{attribute 'GeneratedUsingTerminal: EK1100-0000-0018'}
{attribute addProperty BoxType "EK1100-0000-0018"}
{attribute addProperty Id "Beckhoff_EPP7xxxEK1122Beckhoff_EPP7xxxEK1122_6A0F0FE8478"}
{attribute addProperty CRC "1759912252"}
{attribute addProperty Size "478"}
TYPE Beckhoff_EPP7xxx_68E6213C EXTENDS EK1100_1FC0878B :
STRUCT
	{attribute addProperty Name "Beckhoff_EPP7xxxEK1122"}
	{attribute addProperty PreviousPort "Beckhoff EPP7xxx : B"}
	Beckhoff_EPP7xxxEK1122 : Beckhoff_EPP7xxxEK1122_6A0F0FE8;
END_STRUCT
END_TYPE

(* stored: Version 1.2.0.0, ProductVersion 3.1.4024.9
   DUT Beckhoff_EPP7xxx_68E6213C: Id {2522ea29-0bc9-4fc4-a396-822a9f31a366} *)
